INTERFACE I_LensSet EXTENDS I_Fallible


METHOD GetFocalLengthOf : LREAL
VAR_INPUT
    nLensNum : INT;
END_VAR
END_METHOD


METHOD GetMultiplierOf : INT
VAR_INPUT
    nLensNum : INT;
END_VAR
END_METHOD


PROPERTY NumLenses : INT
GET
END_GET
END_PROPERTY

END_INTERFACE

(* stored: Version 1.1.0.1
   Itf I_LensSet: Id {af8928da-13fc-4163-8eee-ff4c1855e013}
   Method GetFocalLengthOf: Id {a44f57d4-6faf-454a-afd0-8c63627056bd}
   Method GetMultiplierOf: Id {31d62eab-b19c-48ea-b5d4-36044a92d787}
   Property NumLenses: Id {7f9d4f52-506b-44d3-a51f-13e55de73178}
   Get Get: Id {ad7b4714-f6a1-4b3b-9746-9146660d587b} *)
